Staubli VAL3: _DECODE.pgx

public program _decode(string x_sInString, string& x_sOutString[], string x_sBreakChar, num x_nMode)
begin
  // ABSTRACT:
  // Extract part of a string as delimited by break characters
  //
  // INPUT PARMS:
  //  x_sInString    : Input string that will be scanned.
  //  x_sBreakChar   : Break character which are to be considered
  //  x_nValue[]     : Real value to be inserted into the input string
  //  x_nMode        : Control the operation performed by the function
  //      = 0 -->    : Returns the input string in which the characters up to the
  //                 first break character are removed.
  //      = 1 -->  Characters up to the first NONbreak character are removed from the
  //               input string and returned in the outputString
  //
  // OUTPUT PARMS:
  // x_sOutString    : Output String
  //
  //Created 21/12/05                              C.CURRIVAND
  //--------------------------------------------------------------
  // Set default value for break character
  if x_sBreakChar==""
    x_sBreakChar=" "
  endIf
  switch x_nMode
    case 0
      while (mid(x_sInString,1,0)!=x_sBreakChar)
        x_sInString=delete(x_sInString,1,0)
        //? x_sInString
      endWhile
      // remove break character
      x_sOutString=delete(x_sInString,1,0)
    break
    case 1
      while mid(x_sInString,1,0)==x_sBreakChar
        x_sInString=delete(x_sInString,1,0)
        //? x_sInString
      endWhile
      x_sOutString=x_sInString
    break
  endSwitch
end
